// TwinCAT 3 PLC project PLC_1
// ProgramVersion: 3.1.4026.16
// CompilerDefines: VISU_USEPROPERTYINFO
// libraries:
//   Tc2_Standard, * (Beckhoff Automation GmbH)
//   Tc2_System, * (Beckhoff Automation GmbH)
//   VisuSymbols, 4.5.0.0 (System)
// project tree:
//   DUTs/ E_PizzaOvenStates.TcDUT
//   / GlobalTextList.TcGTLO, PlcTask.TcTTO, Visualization Manager.TcVMO (not stored)
//   POUs/ FB_PizzaOven.TcPOU, MAIN.TcPOU
//   VISUs/ Visualization.TcVIS
// real-time tasks:
//   TASK PlcTask: cycle T#10ms, priority 20, ADS port 350

CONFIGURATION PLC_1
    RESOURCE PLC ON TwinCAT3
        TASK PlcTask(INTERVAL := T#10ms, PRIORITY := 20);
        PROGRAM MAIN WITH PlcTask : MAIN;
    END_RESOURCE
END_CONFIGURATION

// ---- DUTs/E_PizzaOvenStates.TcDUT
{attribute 'qualified_only'}
{attribute 'strict'}
{attribute 'to_string'}
TYPE E_PizzaOvenStates :
(
	WaitForPizzaInOven 	:= 0,
	WeJustGotAPizza		:= 1,
	MovePizzaOutOfOven	:= 2,
	MovePizzaToTray		:=3
);
END_TYPE

// ---- POUs/MAIN.TcPOU
PROGRAM MAIN
VAR
	fbPizzaOven : FB_PizzaOven ;
	bLoadPizza				: BOOL; //InsertPizza button
	bRemovePizza			: BOOL; //PackagePizza button
END_VAR

fbPizzaOven(bLoadPizza := bLoadPizza, bRemovePizza := bRemovePizza);

END_PROGRAM

// ---- POUs/FB_PizzaOven.TcPOU
FUNCTION_BLOCK FB_PizzaOven
VAR_INPUT
	bLoadPizza				: BOOL; //InsertPizza button
	bRemovePizza			: BOOL; //PackagePizza button
END_VAR
VAR_OUTPUT
	bBuzzer 				: BOOL;
	nTotalPizzasCooked	: UINT := 0;
END_VAR
VAR
	bPizzaInOven 			: BOOL; //PizzaInOven 	Visual 	
	bPizzaOnDeck			: BOOL; //PizzaOnDeck 	Visual 
	bPizzaDone				: BOOL; //PizzaDone 	Visual
	
	fbTimer : TON ;
	tOvenTime			: TIME := T#4S;
	fbLoad_RTRIG		: R_TRIG;
	fbRemove_RTRIG		: R_TRIG;
	
	sCurrentStateString : STRING ;
	eState 				: E_PizzaOvenStates ;
END_VAR

IF bPizzaOnDeck AND NOT bPizzaInOven THEN
	bPizzaOnDeck := FALSE;
	bPizzaInOven := TRUE ;
END_IF

fbLoad_RTRIG(CLK := bLoadPizza) ;
IF fbLoad_RTRIG.Q THEN
	//bLoadPizza := FALSE ;
	bPizzaOnDeck := TRUE;
END_IF

fbRemove_RTRIG(CLK := bRemovePizza);
IF fbRemove_RTRIG.Q THEN
	//bPizzaDone := FALSE;
	bRemovePizza := FALSE;  
END_IF

// Once program Starts init state is WaitForPizzaInOven
CASE eState OF 
	E_PizzaOvenStates.WaitForPizzaInOven:
		sCurrentStateString := 'WaitForPizzaInOven';
        IF bPizzaInOven THEN
			eState := E_PizzaOvenStates.WeJustGotAPizza;
		END_IF
	// break ;
	
	E_PizzaOvenStates.WeJustGotAPizza:
	sCurrentStateString := 'WeJustGotAPizza';
	// Start the Timer
    fbTimer(IN := TRUE, PT := tOvenTime);
	IF fbTimer.Q THEN
		fbTimer(IN := FALSE);
		eState := E_PizzaOvenStates.MovePizzaOutOfOven;
	END_IF
	// break ;
	
	E_PizzaOvenStates.MovePizzaOutOfOven:
		sCurrentStateString := 'MovePizzaOutOfOven';
		IF NOT bPizzaDone THEN
			bPizzaInOven := FALSE ;
			bPizzaDone := TRUE;
			bBuzzer := FALSE ;
			eState := E_PizzaOvenStates.MovePizzaToTray ;
		ELSE
			bBuzzer := TRUE ;
			sCurrentStateString := 'PizzaIsBurning';
		END_IF
		
	// break ;
	E_PizzaOvenStates.MovePizzaToTray:
		sCurrentStateString := 'MovePizzaToTray';
		nTotalPizzasCooked := nTotalPizzasCooked +1 ;
		eState := E_PizzaOvenStates.WaitForPizzaInOven;
	/// break ;
	
	ELSE 
		sCurrentStateString := 'Invaild State' ;
		
END_CASE

END_FUNCTION_BLOCK

// ---- GlobalTextList.TcGTLO
TEXTLIST GlobalTextList
  458 = '%s'
  926 = 'Buzzer'
  974 = 'Elapsed Time'
  43 = 'Elapsed Time: %s'
  662 = 'Insert Pizza'
  580 = 'Pacakge Pizza'
  670 = 'Pizza'
  804 = 'Pizza On Deck'
  579 = 'Pizza(Done)'
  11 = 'Pizza(On Deck)'
  219 = 'Take Pizza Out'
  987 = 'Total Cooked Pizzas'
  570 = 'Total Cooked Pizzas: %i'
END_TEXTLIST

// ---- VISUs/Visualization.TcVIS
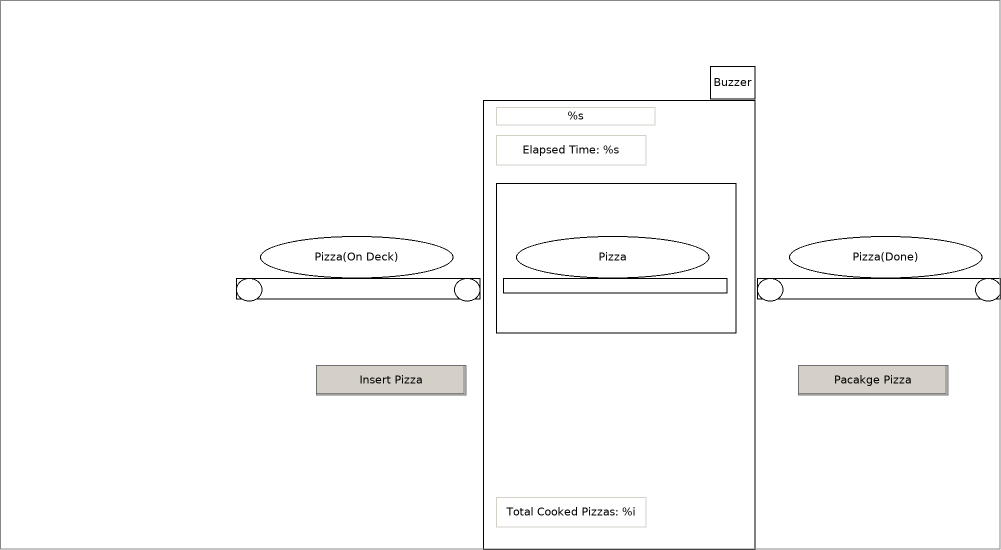
VISUALIZATION Visualization  // 1001x550
    Rectangle (483,100 272x450)
    Button (316,365 150x30), "Insert Pizza"
        tap MAIN.bLoadPizza
        OnMouseClick: execute { MAIN.bPizzaInOven := TRUE ; }
    Button (798,365 150x30), "Pacakge Pizza"
        toggle MAIN.bRemovePizza
        OnMouseClick: execute { MAIN.bPizzaInOven := FALSE }
    Rectangle (496,183 240x150)
    Ellipse (516,236 193x42), "Pizza", invisible if: NOT fbPizzaOven.bPizzaInOven
    Textfield (496,135 150x30), "Elapsed Time: %s", text variable: fbPizzaOven.fbTimer.ET
    Textfield (496,497 150x30), "Total Cooked Pizzas: %i", text variable: FB_PizzaOven.nTotalPizzasCooked
    Rectangle (236,278 244x21)
    Ellipse (236,278 26x23)
    Ellipse (454,278 26x23)
    Rectangle (503,278 224x15)
    Rectangle (757,278 244x21)
    Ellipse (757,278 26x23)
    Ellipse (975,278 26x23)
    Ellipse (260,236 193x42), "Pizza(On Deck)", invisible if: NOT fbPizzaOven.bPizzaOnDeck
    Ellipse (789,236 193x42), "Pizza(Done)", invisible if: NOT fbPizzaOven.bPizzaDone
    Rectangle (710,66 45x33), "Buzzer", colour toggle: fbPizzaOven.bBuzzer
    Textfield (496,107 159x18), "%s", text variable: fbPizzaOven.sCurrentStateString
END_VISUALIZATION
